// TIA Portal V21 export
TYPE "STD"
   STRUCT
      "SET TEMP1" : Real := 0.0;
      "SET TEMP2" : Real := 0.0;
      "SET TEMP3" : Real := 0.0;
      "SET PRESS" : Real := 0.0;
      "SET HOLD1" : Int := 0;
      "SET HOLD2" : Int := 0;
      "SET HOLD3" : Int := 0;
      "SET VCC" : Real := 0.0;
      "SET UP PRESS" : Real := 0.0;
      "SET VCC HOLD" : Int := 0;
      "SET NO OF PULSE" : Int := 0;
   END_STRUCT;
END_TYPE
